// TIA Portal V19 export
DATA_BLOCK "DB_HW"   // DB53
{ S7_Optimized_Access := 'FALSE' }
// stored: AutoNumber false
   VAR RETAIN
      Anzahl : Int := 0;   // * Anzahl der Höhenwechsel
      Offset : Int := 10;   // * Startadresse Einträge
      lengHW : Int := 6;   // * Länge eines Eintrages in Byte
      resW : Int := 0;
      resW1 : Int := 0;
      HW : Array[1..8] of Struct
         Pos : DInt;
         Ebene_rck : Byte;
         Ebene_vor : Byte;
      END_STRUCT;
   END_VAR
BEGIN
   HW[1..8].Pos := 0;
   HW[1..8].Ebene_rck := 16#00;
   HW[1..8].Ebene_vor := 16#00;
END_DATA_BLOCK
